// TIA Portal V19 export
ORGANIZATION_BLOCK "Main"   // OB1, LAD, ProgramCycle
TITLE = "Main Program Sweep (Cycle)"
{ S7_Optimized_Access := 'TRUE' }
// stored: SetENOAutomatically false
   VAR_INPUT
      Initial_Call : Bool;   // Initial call of this OB
      Remanence : Bool;   // =True, if remanent data are available
   END_VAR
   VAR_TEMP   // added for the SCL form of the ladder/FBD networks
      _w1 : Bool;
   END_VAR
BEGIN

REGION Network 1: Control
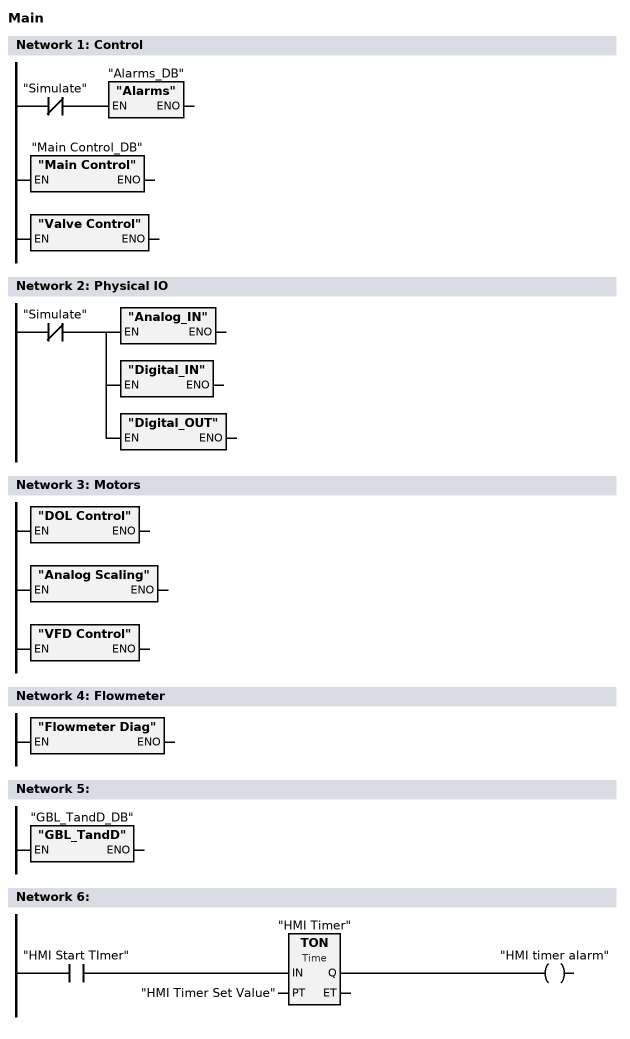
   RUNG wire#powerrail
      I_Contact( "Simulate" )
      "Alarms_DB"()
   END_RUNG
   RUNG wire#powerrail
      "Main Control_DB"()
   END_RUNG
   RUNG wire#powerrail
      "Valve Control"()
   END_RUNG
   // the same network as SCL:
   IF NOT "Simulate" THEN
       "Alarms_DB"();   // "Alarms"
   END_IF;
   "Main Control_DB"();   // "Main Control"
   "Valve Control"();
END_REGION

REGION Network 2: Physical IO
   RUNG wire#powerrail
      I_Contact( "Simulate" )
      wire#w1
      "Analog_IN"()
   END_RUNG
   RUNG wire#w1
      "Digital_IN"()
   END_RUNG
   RUNG wire#w1
      "Digital_OUT"()
   END_RUNG
   // the same network as SCL:
   #_w1 := NOT "Simulate";
   IF #_w1 THEN
       "Analog_IN"();
       "Digital_IN"();
       "Digital_OUT"();
   END_IF;
END_REGION

REGION Network 3: Motors
   RUNG wire#powerrail
      "DOL Control"()
   END_RUNG
   RUNG wire#powerrail
      "Analog Scaling"()
   END_RUNG
   RUNG wire#powerrail
      "VFD Control"()
   END_RUNG
   // the same network as SCL:
   "DOL Control"();
   "Analog Scaling"();
   "VFD Control"();
END_REGION

REGION Network 4: Flowmeter
   RUNG wire#powerrail
      "Flowmeter Diag"()
   END_RUNG
   // the same network as SCL:
   "Flowmeter Diag"();
END_REGION

REGION Network 5
   RUNG wire#powerrail
      "GBL_TandD_DB"()
   END_RUNG
   // the same network as SCL:
   "GBL_TandD_DB"();   // "GBL_TandD"
END_REGION

REGION Network 6
   RUNG wire#powerrail
      Contact( "HMI Start TImer" )
      { S7_Templates := "time_type := Time" } "HMI Timer".TON(pt := "HMI Timer Set Value", et =>)
      Coil( "HMI timer alarm" )
   END_RUNG
   // the same network as SCL:
   "HMI Timer".TON(IN := "HMI Start TImer", PT := "HMI Timer Set Value");
   "HMI timer alarm" := "HMI Timer".Q;
END_REGION
END_ORGANIZATION_BLOCK
